(* PLC project mtcs_dome, Institute of Astronomy OntoManager 0.0.1 *)
(* stored: creationDateTime 2024-08-13T09:19:36.315732, modificationDateTime 2024-08-13T09:19:36.315732 *)

TYPE DomeParts : STRUCT
  shutter : DomeShutter;  (* Shutter mechanism *)
  rotation : DomeRotation;  (* Rotation mechanism *)
  light : DomeLight;  (* Light in dome *)
  io : DomeIO;  (* EtherCAT devices *)
  configManager : ConfigManager;  (* The config manager (to load/save/activate configuration data) *)
END_STRUCT;
END_TYPE

TYPE DomeShutterParts : STRUCT
  pumpsRelay : SimpleRelay;  (* Relay to start the pumps motors *)
  upperOpenRelay : SimpleRelay;  (* Relay to open the upper shutter panel *)
  upperCloseRelay : SimpleRelay;  (* Relay to close the upper shutter panel *)
  lowerOpenRelay : SimpleRelay;  (* Relay to open the upper shutter panel *)
  lowerCloseRelay : SimpleRelay;  (* Relay to close the upper shutter panel *)
END_STRUCT;
END_TYPE

TYPE DomeRotationParts : STRUCT
  masterAxis : AngularAxis;  (* Master axis *)
  slaveAxis : AngularAxis;  (* Slave axis *)
  drive : AX52XXDrive;  (* Dual axis drive *)
END_STRUCT;
END_TYPE

TYPE DomeLightParts : STRUCT
  switchOnRelay : SimpleRelay;  (* Relay to switch on the light *)
END_STRUCT;
END_TYPE

TYPE DomeIOParts : STRUCT
  coupler : EtherCatDevice;  (* Coupler *)
  slot1 : EtherCatDevice;  (* Slot 1 *)
  slot2 : EtherCatDevice;  (* Slot 2 *)
  slot3 : EtherCatDevice;  (* Slot 3 *)
  slot4 : EtherCatDevice;  (* Slot 4 *)
  drive : EtherCatDevice;  (* Drive *)
END_STRUCT;
END_TYPE

TYPE DomeProcesses : STRUCT
  initialize : Process;  (* Start initializing *)
  lock : Process;  (* Lock the cover *)
  unlock : Process;  (* Unlock the cover *)
  changeOperatingState : ChangeOperatingStateProcess;  (* Change the operating state (e.g. AUTO, MANUAL, ...) *)
  reset : Process;  (* Reset any errors *)
  powerOn : Process;  (* Power on the dome *)
  powerOff : Process;  (* Power off the dome *)
  syncWithAxes : Process;  (* Synchronize the dome once with the axes *)
  startTracking : Process;  (* Start tracking the axes *)
  stopTracking : Process;  (* Stop tracking the axes *)
  stop : Process;  (* Stop the rotation movement and/or tracking *)
  moveKnownPosition : DomeMoveKnownPositionProcess;  (* Move the dome to the given known position *)
END_STRUCT;
END_TYPE

TYPE DomeShutterProcesses : STRUCT
  reset : Process;  (* Reset errors *)
  open : Process;  (* Open both panels *)
  close : Process;  (* Close both panels *)
  stop : Process;  (* Stop the panels *)
  lowerOpen : Process;  (* Open the lower panel *)
  lowerClose : Process;  (* Close the lower panel *)
  upperOpen : Process;  (* Open the upper panel *)
  upperClose : Process;  (* Close the upper panel *)
END_STRUCT;
END_TYPE

TYPE DomeRotationProcesses : STRUCT
  reset : Process;  (* Reset errors *)
  stop : Process;  (* Stop the rotation *)
  moveAbsolute : DomeMoveProcess;  (* Move absolute *)
  moveRelative : DomeMoveProcess;  (* Move relative *)
  home : Process;  (* Perform a homing *)
  powerOn : Process;  (* Power on master and slave *)
  powerOff : Process;  (* Power off master and slave *)
END_STRUCT;
END_TYPE

TYPE DomeLightProcesses : STRUCT
  reset : Process;  (* Reset errors *)
  switchLightOn : Process;  (* Turn On the light in the dome *)
  switchLightOff : Process;  (* Turn Off the light in the dome *)
END_STRUCT;
END_TYPE

TYPE DomeStatuses : STRUCT
  initializationStatus : InitializationStatus;
  healthStatus : HealthStatus;
  busyStatus : BusyStatus;
  operatingStatus : OperatingStatus;
  poweredStatus : PoweredStatus;
END_STRUCT;
END_TYPE

TYPE DomeShutterStatuses : STRUCT
  apertureStatus : ApertureStatus;  (* Combined aperture status (i.e. of both panels) *)
  lowerApertureStatus : ApertureStatus;  (* Aperture status of the lower panel *)
  upperApertureStatus : ApertureStatus;  (* Aperture status of the upper panel *)
  healthStatus : HealthStatus;  (* Health status *)
  busyStatus : BusyStatus;  (* Busy status *)
END_STRUCT;
END_TYPE

TYPE DomeRotationStatuses : STRUCT
  healthStatus : HealthStatus;  (* Health status *)
  busyStatus : BusyStatus;  (* Busy status *)
  poweredStatus : PoweredStatus;  (* Powered status *)
END_STRUCT;
END_TYPE

TYPE DomeLightStatuses : STRUCT
  healthStatus : HealthStatus;  (* Health status *)
  busyStatus : BusyStatus;  (* Busy status *)
END_STRUCT;
END_TYPE

TYPE DomeIOStatuses : STRUCT
  healthStatus : HealthStatus;  (* Is the I/O in a healthy state? *)
END_STRUCT;
END_TYPE

TYPE DomeConfig : STRUCT
  shutter : DomeShutterConfig;  (* The config of the shutter mechanism *)
  rotation : DomeRotationConfig;  (* The config of the rotation system *)
  light : DomeLightConfig;  (* The config of the light in the dome *)
  maxTrackingDistance : LREAL;  (* The maximum distance between telescope and dome while tracking *)
  trackingLoopTime : LREAL;  (* Loop time, in seconds, of the tracking. *)
  knownPositions : DomeKnownPositionsConfig;  (* The known positions of the dome *)
  knownPositionTolerance : LREAL;  (* Tolerance (in degrees) to determine if the dome is at a known position *)
END_STRUCT;
END_TYPE

TYPE DomeKnownPositionConfig : STRUCT
  name : STRING;  (* The name of the position (e.g. 'PARK') *)
  position : LREAL;  (* Azimuth in degrees *)
END_STRUCT;
END_TYPE

TYPE DomeKnownPositionsConfig : STRUCT
  position0 : DomeKnownPositionConfig;  (* Known position 0 *)
  position1 : DomeKnownPositionConfig;  (* Known position 1 *)
  position2 : DomeKnownPositionConfig;  (* Known position 2 *)
  position3 : DomeKnownPositionConfig;  (* Known position 3 *)
  position4 : DomeKnownPositionConfig;  (* Known position 4 *)
  position5 : DomeKnownPositionConfig;  (* Known position 5 *)
  position6 : DomeKnownPositionConfig;  (* Known position 6 *)
  position7 : DomeKnownPositionConfig;  (* Known position 7 *)
  position8 : DomeKnownPositionConfig;  (* Known position 8 *)
  position9 : DomeKnownPositionConfig;  (* Known position 9 *)
END_STRUCT;
END_TYPE

TYPE DomeShutterConfig : STRUCT
  wirelessPolling : LREAL;  (* Polling frequency of the wireless I/O device, in seconds. Negative value = no polling. *)
  wirelessIpAddress : STRING;  (* IP address of the wireless I/O device *)
  wirelessPort : UINT;  (* Port of the wireless I/O device *)
  wirelessUnitID : USINT;  (* Unit ID the wireless I/O device *)
  wirelessTimeoutSeconds : LREAL;  (* The timeout of a single command. Does not lead to an error (yet), because we still retry. *)
  wirelessRetriesSeconds : LREAL;  (* The total timeout of the retries. If no valid data is received after this time, then we consider the shutters in error. *)
  upperEstimatedOpenTime : LREAL;  (* Estimated opening time of the upper panel, in seconds *)
  upperEstimatedCloseTime : LREAL;  (* Estimated closing time of the upper panel, in seconds *)
  lowerEstimatedOpenTime : LREAL;  (* Estimated opening time of the lower panel, in seconds *)
  lowerEstimatedCloseTime : LREAL;  (* Estimated closing time of the lower panel, in seconds *)
  lowerOpenTimeout : LREAL;  (* Opening timeout of the lower panel, in seconds *)
  lowerCloseTimeout : LREAL;  (* Closing timeout of the lower panel, in seconds *)
  upperOpenTimeout : LREAL;  (* Opening timeout of the upper panel, in seconds *)
  upperCloseTimeout : LREAL;  (* Closing timeout of the upper panel, in seconds *)
  timeAfterStop : LREAL;  (* Time to wait after a stop command, in seconds *)
END_STRUCT;
END_TYPE

TYPE DomeRotationConfig : STRUCT
  maxMovingVelocity : LREAL;  (* Maximum velocity when moving absolute or relative, in degrees per second *)
  maxMasterSlaveLag : LREAL;  (* Below this lag value (in degrees), the lag is considered not an error *)
  torqueCoefficientV : LREAL;  (* Coefficient v in 'SlaveTorque = v * MasterVelo + a * MasterAcceleration *)
  torqueCoefficientA : LREAL;  (* Coefficient a in 'SlaveTorque = v * MasterVelo + a * MasterAcceleration *)
  homePosition : LREAL;  (* Azimuth position of the home sensor, in degrees *)
  homingMoveOutOfSensorDistance : LREAL;  (* If on the sensor, move this distance, in degrees *)
  homingStage1Velocity : LREAL;  (* Velocity, in degrees per second, of the first homing stage *)
  homingStage1Timeout : LREAL;  (* Timeout of the first homing stage, in seconds *)
  homingStage2Velocity : LREAL;  (* Velocity, in degrees per second, of the second homing stage *)
  homingStage2Timeout : LREAL;  (* Timeout of the second homing stage, in seconds *)
  homingDoTwoStages : BOOL;  (* True for 2-stages homing, False for 1-stage homing. *)
  quickStopDeceleration : LREAL;  (* Quick stop deceleration, in degrees/sec2 *)
  quickStopJerk : LREAL;  (* Quick stop jerk, in degrees/sec3 *)
END_STRUCT;
END_TYPE

TYPE DomeLightConfig : STRUCT
  timeDomeLightOn : LREAL;  (* Time to keep the light on, in seconds *)
  enableDomeLight : BOOL;  (* True for enabling the control of the light *)
END_STRUCT;
END_TYPE

TYPE DomeMoveKnownPositionProcessArgs : STRUCT
  name : STRING;  (* Name of the position to move to *)
END_STRUCT;
END_TYPE

TYPE DomeMoveProcessArgs : STRUCT
  position : LREAL;  (* New absolute or relative position value in degrees *)
END_STRUCT;
END_TYPE

FUNCTION_BLOCK SM_Dome
  VAR_INPUT
    {attribute 'OPC.UA.DA' := '1'}
    {attribute 'OPC.UA.DA.Access' := '1'}
    editableConfig : DomeConfig;  (* Editable configuration of the cover *)
  END_VAR
  VAR_OUTPUT
    {attribute 'OPC.UA.DA' := '1'}
    {attribute 'OPC.UA.DA.Access' := '1'}
    actualStatus : STRING;  (* Current status description *)
    previousStatus : STRING;  (* Previous status description *)
    {attribute 'OPC.UA.DA' := '1'}
    {attribute 'OPC.UA.DA.Access' := '1'}
    config : DomeConfig;  (* Active configuration of the cover *)
    {attribute 'OPC.UA.DA' := '1'}
    {attribute 'OPC.UA.DA.Access' := '1'}
    isPoweredOffByPersonInDome : BOOL;  (* True if the dome is powered off due to a person entering the dome *)
    {attribute 'OPC.UA.DA' := '1'}
    {attribute 'OPC.UA.DA.Access' := '1'}
    isTracking : BOOL;  (* True if the dome is tracking the telescope *)
    {attribute 'OPC.UA.DA' := '1'}
    {attribute 'OPC.UA.DA.Access' := '1'}
    telescopeTargetDistance : AngularPosition;  (* Actual distance between telescope target and dome *)
    {attribute 'OPC.UA.DA' := '1'}
    {attribute 'OPC.UA.DA.Access' := '1'}
    isAtKnownPosition : BOOL;  (* True if the dome is at a known position *)
    {attribute 'OPC.UA.DA' := '1'}
    {attribute 'OPC.UA.DA.Access' := '1'}
    actualKnownPositionName : STRING;  (* Name of the known position if isAtKnownPosition is True *)
    statuses : DomeStatuses;  (* Statuses of the state machine *)
    parts : DomeParts;  (* Parts of the state machine *)
    processes : DomeProcesses;  (* Processes of the state machine *)
  END_VAR
  VAR_IN_OUT
    {attribute 'OPC.UA.DA' := '0'}
    operatorStatus : OperatorStatus;  (* Reference to the operator (observer/tech) *)
    {attribute 'OPC.UA.DA' := '0'}
    activityStatus : ActivityStatus;  (* Shared activity status *)
    {attribute 'OPC.UA.DA' := '0'}
    aziTargetPos : AngularPosition;  (* Azimuth target position of the telescope Axes *)
    {attribute 'OPC.UA.DA' := '0'}
    safetyDomeShutter : SafetyDomeShutter;  (* Reference to the dome shutter safety *)
    {attribute 'OPC.UA.DA' := '0'}
    safetyMotionBlocking : SafetyMotionBlocking;  (* Reference to the motion blocking safety *)
    {attribute 'OPC.UA.DA' := '0'}
    safetyDomeAccess : SafetyDomeAccess;  (* Reference to the dome access safety *)
  END_VAR

            parts.shutter(
    initializationStatus := statuses.initializationStatus,
    operatorStatus := operatorStatus,
    operatingStatus := statuses.operatingStatus,
    activityStatus := activityStatus,
    safety := safetyDomeShutter,
    config := config.shutter);
parts.rotation(
    initializationStatus := statuses.initializationStatus,
    operatorStatus := operatorStatus,
    operatingStatus := statuses.operatingStatus,
    config := config.rotation);
parts.light(
    initializationStatus := statuses.initializationStatus,
    operatorStatus := operatorStatus,
    operatingStatus := statuses.operatingStatus,
    activityStatus := activityStatus,
    config := config.light);
parts.io();
parts.configManager( isEnabled := operatorStatus.tech );
statuses.initializationStatus();
statuses.healthStatus(
    isGood := parts.shutter.statuses.healthStatus.isGood AND (parts.rotation.statuses.healthStatus.isGood AND (parts.light.statuses.healthStatus.isGood AND parts.io.statuses.healthStatus.isGood)),
    hasWarning := parts.shutter.statuses.healthStatus.hasWarning OR (parts.rotation.statuses.healthStatus.hasWarning OR (parts.light.statuses.healthStatus.hasWarning OR parts.io.statuses.healthStatus.hasWarning)));
statuses.busyStatus( isBusy := parts.shutter.statuses.busyStatus.busy OR parts.rotation.statuses.busyStatus.busy );
statuses.operatingStatus( superState := statuses.initializationStatus.initialized );
statuses.poweredStatus( isEnabled := parts.rotation.statuses.poweredStatus.enabled );
processes.initialize( isEnabled := (NOT(statuses.initializationStatus.locked)) AND (statuses.initializationStatus.shutdown OR (statuses.initializationStatus.initializingFailed OR statuses.initializationStatus.initialized)) );
processes.lock( isEnabled := operatorStatus.tech );
processes.unlock( isEnabled := operatorStatus.tech AND statuses.initializationStatus.locked );
processes.changeOperatingState( isEnabled := FALSE );
processes.reset( isEnabled := statuses.busyStatus.idle AND statuses.initializationStatus.initialized );
processes.powerOn( isEnabled := (NOT(statuses.initializationStatus.locked)) AND (statuses.initializationStatus.initialized AND processes.powerOn.statuses.busyStatus.idle) );
processes.powerOff( isEnabled := statuses.initializationStatus.initialized AND processes.powerOff.statuses.busyStatus.idle );
processes.syncWithAxes( isEnabled := statuses.initializationStatus.initialized AND (statuses.busyStatus.idle AND (statuses.poweredStatus.enabled AND parts.rotation.isHomed)) );
processes.startTracking( isEnabled := statuses.poweredStatus.enabled AND ((NOT(isTracking)) AND parts.rotation.isHomed) );
processes.stopTracking( isEnabled := isTracking );
processes.stop( isEnabled := statuses.busyStatus.busy OR (isTracking OR operatorStatus.tech) );
processes.moveKnownPosition( isEnabled := statuses.initializationStatus.initialized AND (statuses.busyStatus.idle AND (statuses.poweredStatus.enabled AND parts.rotation.isHomed)) );

          

{attribute 'TcRpcEnable' := '1'}
METHOD initialize : RequestResults
                  initialize := THIS^.processes.initialize.request();

                
END_METHOD

{attribute 'TcRpcEnable' := '1'}
METHOD lock : RequestResults
                  lock := THIS^.processes.lock.request();

                
END_METHOD

{attribute 'TcRpcEnable' := '1'}
METHOD unlock : RequestResults
                  unlock := THIS^.processes.unlock.request();

                
END_METHOD

{attribute 'TcRpcEnable' := '1'}
METHOD changeOperatingState : RequestResults
  VAR_INPUT
    state : OperatingStates;
  END_VAR
                  changeOperatingState := THIS^.processes.changeOperatingState.request( state := state );

                
END_METHOD

{attribute 'TcRpcEnable' := '1'}
METHOD reset : RequestResults
                  reset := THIS^.processes.reset.request();

                
END_METHOD

{attribute 'TcRpcEnable' := '1'}
METHOD powerOn : RequestResults
                  powerOn := THIS^.processes.powerOn.request();

                
END_METHOD

{attribute 'TcRpcEnable' := '1'}
METHOD powerOff : RequestResults
                  powerOff := THIS^.processes.powerOff.request();

                
END_METHOD

{attribute 'TcRpcEnable' := '1'}
METHOD syncWithAxes : RequestResults
                  syncWithAxes := THIS^.processes.syncWithAxes.request();

                
END_METHOD

{attribute 'TcRpcEnable' := '1'}
METHOD startTracking : RequestResults
                  startTracking := THIS^.processes.startTracking.request();

                
END_METHOD

{attribute 'TcRpcEnable' := '1'}
METHOD stopTracking : RequestResults
                  stopTracking := THIS^.processes.stopTracking.request();

                
END_METHOD

{attribute 'TcRpcEnable' := '1'}
METHOD stop : RequestResults
                  stop := THIS^.processes.stop.request();

                
END_METHOD

{attribute 'TcRpcEnable' := '1'}
METHOD moveKnownPosition : RequestResults
  VAR_INPUT
    name : STRING;
  END_VAR
                  moveKnownPosition := THIS^.processes.moveKnownPosition.request( name := name );

                
END_METHOD

{attribute 'TcRpcEnable' := '1'}
METHOD _log : BOOL
  VAR_INPUT
    name : STRING;  (* Name of this function block instance *)
  END_VAR
  VAR_IN_OUT
    buffer : LogBuffer;  (* Buffer to write all logging to *)
  END_VAR
  VAR
    subBuffer : LogBuffer;  (* Temporary buffer to write logging by parts (sub-statemachines) to *)
  END_VAR
                  THIS^.parts.shutter._log(
    name := 'shutter',
    buffer := subBuffer);
THIS^.parts.rotation._log(
    name := 'rotation',
    buffer := subBuffer);
THIS^.parts.light._log(
    name := 'light',
    buffer := subBuffer);
THIS^.parts.io._log(
    name := 'io',
    buffer := subBuffer);
THIS^.parts.configManager._log(
    name := 'configManager',
    buffer := subBuffer);
THIS^.processes.initialize._log(
    name := 'processes.initialize',
    buffer := subBuffer);
THIS^.processes.lock._log(
    name := 'processes.lock',
    buffer := subBuffer);
THIS^.processes.unlock._log(
    name := 'processes.unlock',
    buffer := subBuffer);
THIS^.processes.changeOperatingState._log(
    name := 'processes.changeOperatingState',
    buffer := subBuffer);
THIS^.processes.reset._log(
    name := 'processes.reset',
    buffer := subBuffer);
THIS^.processes.powerOn._log(
    name := 'processes.powerOn',
    buffer := subBuffer);
THIS^.processes.powerOff._log(
    name := 'processes.powerOff',
    buffer := subBuffer);
THIS^.processes.syncWithAxes._log(
    name := 'processes.syncWithAxes',
    buffer := subBuffer);
THIS^.processes.startTracking._log(
    name := 'processes.startTracking',
    buffer := subBuffer);
THIS^.processes.stopTracking._log(
    name := 'processes.stopTracking',
    buffer := subBuffer);
THIS^.processes.stop._log(
    name := 'processes.stop',
    buffer := subBuffer);
THIS^.processes.moveKnownPosition._log(
    name := 'processes.moveKnownPosition',
    buffer := subBuffer);
LOGGER(
    name := name,
    actualStatus := THIS^.actualStatus,
    previousStatus := THIS^.previousStatus,
    buffer := buffer,
    subBuffer := subBuffer,
    pHealthStatus := ADR(THIS^.statuses.healthStatus),
    pBusyStatus := ADR(THIS^.statuses.busyStatus));

                
END_METHOD
END_FUNCTION_BLOCK

FUNCTION_BLOCK SM_DomeShutter
  VAR_INPUT
    {attribute 'OPC.UA.DA' := '1'}
    {attribute 'OPC.UA.DA.Access' := '1'}
    lowerOpenSignal : BOOL;  (* False if the signal is not present OR if there is a communication error *)
    {attribute 'OPC.UA.DA' := '1'}
    {attribute 'OPC.UA.DA.Access' := '1'}
    lowerClosedSignal : BOOL;  (* False if the signal is not present OR if there is a communication error *)
    {attribute 'OPC.UA.DA' := '1'}
    {attribute 'OPC.UA.DA.Access' := '1'}
    upperOpenSignal : BOOL;  (* False if the signal is not present OR if there is a communication error *)
    {attribute 'OPC.UA.DA' := '1'}
    {attribute 'OPC.UA.DA.Access' := '1'}
    upperClosedSignal : BOOL;  (* False if the signal is not present OR if there is a communication error *)
    {attribute 'OPC.UA.DA' := '1'}
    {attribute 'OPC.UA.DA.Access' := '1'}
    wirelessTimeout : BOOL;  (* True if the wireless communication to the shutter signals is timing out *)
    {attribute 'OPC.UA.DA' := '1'}
    {attribute 'OPC.UA.DA.Access' := '1'}
    wirelessError : BOOL;  (* True if the wireless communication to the shutter signals is in error (other than timeout) *)
    {attribute 'OPC.UA.DA' := '1'}
    {attribute 'OPC.UA.DA.Access' := '1'}
    wirelessErrorId : UDINT;  (* The error id if wirelessError is true *)
    {attribute 'OPC.UA.DA' := '1'}
    {attribute 'OPC.UA.DA.Access' := '1'}
    wirelessData : UINT;  (* The received wireless data *)
    {attribute 'OPC.UA.DA' := '1'}
    {attribute 'OPC.UA.DA.Access' := '1'}
    upperTimeRemaining : Duration;  (* Estimated time remaining to open/close the upper panel *)
    {attribute 'OPC.UA.DA' := '1'}
    {attribute 'OPC.UA.DA.Access' := '1'}
    lowerTimeRemaining : Duration;  (* Estimated time remaining to open/close the lower panel *)
    {attribute 'OPC.UA.DA' := '1'}
    {attribute 'OPC.UA.DA.Access' := '1'}
    isLowerMonitored : BOOL;  (* TRUE if the lower shutter panel is being monitored *)
    {attribute 'OPC.UA.DA' := '1'}
    {attribute 'OPC.UA.DA.Access' := '1'}
    noOfLowerAutoClosings : INT;  (* The number of times that the lower panel has been closed automatically, by monitoring *)
    {attribute 'OPC.UA.DA' := '1'}
    {attribute 'OPC.UA.DA.Access' := '1'}
    manualOpenUpper AT %I* : BOOL;  (* Manual operation: open upper switch *)
    {attribute 'OPC.UA.DA' := '1'}
    {attribute 'OPC.UA.DA.Access' := '1'}
    manualCloseUpper AT %I* : BOOL;  (* Manual operation: close upper switch *)
    {attribute 'OPC.UA.DA' := '1'}
    {attribute 'OPC.UA.DA.Access' := '1'}
    manualOpenLower AT %I* : BOOL;  (* Manual operation: open lower switch *)
    {attribute 'OPC.UA.DA' := '1'}
    {attribute 'OPC.UA.DA.Access' := '1'}
    manualCloseLower AT %I* : BOOL;  (* Manual operation: close lower switch *)
    {attribute 'OPC.UA.DA' := '1'}
    {attribute 'OPC.UA.DA.Access' := '1'}
    manualPumpOn AT %I* : BOOL;  (* Manual operation: pump ON *)
    {attribute 'OPC.UA.DA' := '1'}
    {attribute 'OPC.UA.DA.Access' := '1'}
    automaticOperation AT %I* : BOOL;  (* TRUE if switch is on Auto, FALSE if switch is Manual *)
  END_VAR
  VAR_OUTPUT
    {attribute 'OPC.UA.DA' := '1'}
    {attribute 'OPC.UA.DA.Access' := '1'}
    actualStatus : STRING;  (* Current status description *)
    previousStatus : STRING;  (* Previous status description *)
    statuses : DomeShutterStatuses;  (* Statuses of the state machine *)
    parts : DomeShutterParts;  (* Parts of the state machine *)
    processes : DomeShutterProcesses;  (* Processes of the state machine *)
  END_VAR
  VAR_IN_OUT
    {attribute 'OPC.UA.DA' := '0'}
    initializationStatus : InitializationStatus;  (* Dome initialization status (initialized/initializing/...) *)
    {attribute 'OPC.UA.DA' := '0'}
    operatorStatus : OperatorStatus;  (* MTCS operator (observer/tech) *)
    {attribute 'OPC.UA.DA' := '0'}
    operatingStatus : OperatingStatus;  (* Dome operating status (manual/auto) *)
    {attribute 'OPC.UA.DA' := '0'}
    activityStatus : ActivityStatus;  (* Shared activity status *)
    {attribute 'OPC.UA.DA' := '0'}
    safety : SafetyDomeShutter;  (* The dome shutter safety *)
    {attribute 'OPC.UA.DA' := '0'}
    config : DomeShutterConfig;  (* The shutter config *)
  END_VAR

            parts.pumpsRelay( isEnabled := operatorStatus.tech );
parts.upperOpenRelay( isEnabled := operatorStatus.tech );
parts.upperCloseRelay( isEnabled := operatorStatus.tech );
parts.lowerOpenRelay( isEnabled := operatorStatus.tech );
parts.lowerCloseRelay( isEnabled := operatorStatus.tech );
statuses.apertureStatus(
    superState := NOT(wirelessTimeout OR wirelessError),
    isOpen := statuses.lowerApertureStatus.open AND statuses.upperApertureStatus.open,
    isClosed := statuses.lowerApertureStatus.closed AND statuses.upperApertureStatus.closed);
statuses.lowerApertureStatus(
    superState := NOT(wirelessTimeout OR wirelessError),
    isOpen := lowerOpenSignal,
    isClosed := lowerClosedSignal);
statuses.upperApertureStatus(
    superState := NOT(wirelessTimeout OR wirelessError),
    isOpen := upperOpenSignal,
    isClosed := upperClosedSignal);
statuses.healthStatus(
    isGood := (NOT(wirelessTimeout OR wirelessError)) AND (processes.reset.statuses.healthStatus.isGood AND (processes.open.statuses.healthStatus.isGood AND (processes.close.statuses.healthStatus.isGood AND (processes.stop.statuses.healthStatus.isGood AND (processes.lowerOpen.statuses.healthStatus.isGood AND (processes.lowerClose.statuses.healthStatus.isGood AND (processes.upperOpen.statuses.healthStatus.isGood AND processes.upperClose.statuses.healthStatus.isGood))))))),
    hasWarning := (processes.reset.statuses.healthStatus.hasWarning OR (processes.open.statuses.healthStatus.hasWarning OR (processes.close.statuses.healthStatus.hasWarning OR (processes.stop.statuses.healthStatus.hasWarning OR (processes.lowerOpen.statuses.healthStatus.hasWarning OR (processes.lowerClose.statuses.healthStatus.hasWarning OR (processes.upperOpen.statuses.healthStatus.hasWarning OR processes.upperClose.statuses.healthStatus.hasWarning))))))) OR ((statuses.busyStatus.idle AND statuses.lowerApertureStatus.partiallyOpen) OR ((statuses.busyStatus.idle AND statuses.upperApertureStatus.partiallyOpen) OR (NOT(automaticOperation)))));
statuses.busyStatus( isBusy := processes.reset.statuses.busyStatus.busy OR (processes.open.statuses.busyStatus.busy OR (processes.close.statuses.busyStatus.busy OR (processes.stop.statuses.busyStatus.busy OR (processes.lowerOpen.statuses.busyStatus.busy OR (processes.lowerClose.statuses.busyStatus.busy OR (processes.upperOpen.statuses.busyStatus.busy OR processes.upperClose.statuses.busyStatus.busy)))))) );
processes.reset( isEnabled := TRUE );
processes.open( isEnabled := statuses.healthStatus.isGood AND ((NOT(initializationStatus.locked)) AND (operatorStatus.tech OR (statuses.busyStatus.idle AND (initializationStatus.initialized AND (activityStatus.awake OR activityStatus.moving))))) );
processes.close( isEnabled := statuses.healthStatus.isGood AND ((NOT(initializationStatus.locked)) AND (statuses.busyStatus.idle AND initializationStatus.initialized)) );
processes.stop( isEnabled := statuses.busyStatus.busy );
processes.lowerOpen( isEnabled := processes.open.isEnabled );
processes.lowerClose( isEnabled := processes.close.isEnabled );
processes.upperOpen( isEnabled := processes.open.isEnabled );
processes.upperClose( isEnabled := processes.close.isEnabled );

          

{attribute 'TcRpcEnable' := '1'}
METHOD reset : RequestResults
                  reset := THIS^.processes.reset.request();

                
END_METHOD

{attribute 'TcRpcEnable' := '1'}
METHOD open : RequestResults
                  open := THIS^.processes.open.request();

                
END_METHOD

{attribute 'TcRpcEnable' := '1'}
METHOD close : RequestResults
                  close := THIS^.processes.close.request();

                
END_METHOD

{attribute 'TcRpcEnable' := '1'}
METHOD stop : RequestResults
                  stop := THIS^.processes.stop.request();

                
END_METHOD

{attribute 'TcRpcEnable' := '1'}
METHOD lowerOpen : RequestResults
                  lowerOpen := THIS^.processes.lowerOpen.request();

                
END_METHOD

{attribute 'TcRpcEnable' := '1'}
METHOD lowerClose : RequestResults
                  lowerClose := THIS^.processes.lowerClose.request();

                
END_METHOD

{attribute 'TcRpcEnable' := '1'}
METHOD upperOpen : RequestResults
                  upperOpen := THIS^.processes.upperOpen.request();

                
END_METHOD

{attribute 'TcRpcEnable' := '1'}
METHOD upperClose : RequestResults
                  upperClose := THIS^.processes.upperClose.request();

                
END_METHOD

{attribute 'TcRpcEnable' := '1'}
METHOD _log : BOOL
  VAR_INPUT
    name : STRING;  (* Name of this function block instance *)
  END_VAR
  VAR_IN_OUT
    buffer : LogBuffer;  (* Buffer to write all logging to *)
  END_VAR
  VAR
    subBuffer : LogBuffer;  (* Temporary buffer to write logging by parts (sub-statemachines) to *)
  END_VAR
                  THIS^.parts.pumpsRelay._log(
    name := 'pumpsRelay',
    buffer := subBuffer);
THIS^.parts.upperOpenRelay._log(
    name := 'upperOpenRelay',
    buffer := subBuffer);
THIS^.parts.upperCloseRelay._log(
    name := 'upperCloseRelay',
    buffer := subBuffer);
THIS^.parts.lowerOpenRelay._log(
    name := 'lowerOpenRelay',
    buffer := subBuffer);
THIS^.parts.lowerCloseRelay._log(
    name := 'lowerCloseRelay',
    buffer := subBuffer);
THIS^.processes.reset._log(
    name := 'processes.reset',
    buffer := subBuffer);
THIS^.processes.open._log(
    name := 'processes.open',
    buffer := subBuffer);
THIS^.processes.close._log(
    name := 'processes.close',
    buffer := subBuffer);
THIS^.processes.stop._log(
    name := 'processes.stop',
    buffer := subBuffer);
THIS^.processes.lowerOpen._log(
    name := 'processes.lowerOpen',
    buffer := subBuffer);
THIS^.processes.lowerClose._log(
    name := 'processes.lowerClose',
    buffer := subBuffer);
THIS^.processes.upperOpen._log(
    name := 'processes.upperOpen',
    buffer := subBuffer);
THIS^.processes.upperClose._log(
    name := 'processes.upperClose',
    buffer := subBuffer);
LOGGER(
    name := name,
    actualStatus := THIS^.actualStatus,
    previousStatus := THIS^.previousStatus,
    buffer := buffer,
    subBuffer := subBuffer,
    pHealthStatus := ADR(THIS^.statuses.healthStatus),
    pBusyStatus := ADR(THIS^.statuses.busyStatus));

                
END_METHOD
END_FUNCTION_BLOCK

FUNCTION_BLOCK SM_DomeRotation
  VAR_OUTPUT
    {attribute 'OPC.UA.DA' := '1'}
    {attribute 'OPC.UA.DA.Access' := '1'}
    actualStatus : STRING;  (* Current status description *)
    previousStatus : STRING;  (* Previous status description *)
    {attribute 'OPC.UA.DA' := '1'}
    {attribute 'OPC.UA.DA.Access' := '1'}
    actPos : AngularPosition;  (* The actual position (same as parts.masterAxis!) *)
    {attribute 'OPC.UA.DA' := '1'}
    {attribute 'OPC.UA.DA.Access' := '1'}
    actVelo : AngularVelocity;  (* The actual velocity (same as parts.masterAxis!) *)
    {attribute 'OPC.UA.DA' := '1'}
    {attribute 'OPC.UA.DA.Access' := '1'}
    actTorqueMaster : Torque;  (* The actual torque on the telescope axis by the master motor *)
    {attribute 'OPC.UA.DA' := '1'}
    {attribute 'OPC.UA.DA.Access' := '1'}
    actTorqueSlave : Torque;  (* The actual torque on the telescope axis by the slave motor *)
    {attribute 'OPC.UA.DA' := '1'}
    {attribute 'OPC.UA.DA.Access' := '1'}
    masterSlaveLag : AngularPosition;  (* masterAxis.actPos - slaveAxis.actPos *)
    {attribute 'OPC.UA.DA' := '1'}
    {attribute 'OPC.UA.DA.Access' := '1'}
    masterSlaveLagError : BOOL;  (* (ABS(masterSlaveLag) >= config.maxMasterSlaveLag) AND isHomed AND poweredOn *)
    {attribute 'OPC.UA.DA' := '1'}
    {attribute 'OPC.UA.DA.Access' := '1'}
    homingSensorSignal : BOOL;  (* True = at home position *)
    {attribute 'OPC.UA.DA' := '1'}
    {attribute 'OPC.UA.DA.Access' := '1'}
    isHomed : BOOL;  (* True if homing was done *)
    statuses : DomeRotationStatuses;  (* Statuses of the state machine *)
    parts : DomeRotationParts;  (* Parts of the state machine *)
    processes : DomeRotationProcesses;  (* Processes of the state machine *)
  END_VAR
  VAR_IN_OUT
    {attribute 'OPC.UA.DA' := '0'}
    initializationStatus : InitializationStatus;  (* Reference to the MTCS initialization status *)
    {attribute 'OPC.UA.DA' := '0'}
    operatorStatus : OperatorStatus;  (* Reference to the MTCS operator status *)
    {attribute 'OPC.UA.DA' := '0'}
    operatingStatus : OperatingStatus;  (* Reference to the Dome operating status *)
    {attribute 'OPC.UA.DA' := '0'}
    config : DomeRotationConfig;  (* Reference to the rotation config *)
  END_VAR

            parts.masterAxis( isEnabled := (NOT(initializationStatus.locked)) AND operatorStatus.tech );
parts.slaveAxis( isEnabled := (NOT(initializationStatus.locked)) AND operatorStatus.tech );
parts.drive( isEnabled := (NOT(initializationStatus.locked)) AND operatorStatus.tech );
statuses.healthStatus(
    isGood := (parts.masterAxis.statuses.healthStatus.isGood AND (parts.slaveAxis.statuses.healthStatus.isGood AND (parts.drive.statuses.healthStatus.isGood AND (processes.reset.statuses.healthStatus.isGood AND processes.stop.statuses.healthStatus.isGood)))) AND ((NOT(masterSlaveLagError)) AND (isHomed OR (NOT(initializationStatus.initialized)))),
    hasWarning := parts.masterAxis.statuses.healthStatus.hasWarning OR (parts.slaveAxis.statuses.healthStatus.hasWarning OR (parts.drive.statuses.healthStatus.hasWarning OR (processes.reset.statuses.healthStatus.hasWarning OR processes.stop.statuses.healthStatus.hasWarning))));
statuses.busyStatus( isBusy := parts.masterAxis.statuses.busyStatus.busy OR (parts.slaveAxis.statuses.busyStatus.busy OR (parts.drive.statuses.busyStatus.busy OR (processes.reset.statuses.busyStatus.busy OR processes.stop.statuses.busyStatus.busy))) );
statuses.poweredStatus( isEnabled := parts.masterAxis.statuses.poweredStatus.enabled AND parts.slaveAxis.statuses.poweredStatus.enabled );
processes.reset( isEnabled := statuses.busyStatus.idle );
processes.stop( isEnabled := statuses.busyStatus.busy OR operatorStatus.tech );
processes.moveAbsolute( isEnabled := statuses.busyStatus.idle AND statuses.poweredStatus.enabled );
processes.moveRelative( isEnabled := processes.moveAbsolute.isEnabled );
processes.home( isEnabled := processes.moveAbsolute.isEnabled );
processes.powerOn( isEnabled := (NOT(initializationStatus.locked)) AND statuses.busyStatus.idle );
processes.powerOff( isEnabled := statuses.busyStatus.idle );

          

{attribute 'TcRpcEnable' := '1'}
METHOD reset : RequestResults
                  reset := THIS^.processes.reset.request();

                
END_METHOD

{attribute 'TcRpcEnable' := '1'}
METHOD stop : RequestResults
                  stop := THIS^.processes.stop.request();

                
END_METHOD

{attribute 'TcRpcEnable' := '1'}
METHOD moveAbsolute : RequestResults
  VAR_INPUT
    position : LREAL;
  END_VAR
                  moveAbsolute := THIS^.processes.moveAbsolute.request( position := position );

                
END_METHOD

{attribute 'TcRpcEnable' := '1'}
METHOD moveRelative : RequestResults
  VAR_INPUT
    position : LREAL;
  END_VAR
                  moveRelative := THIS^.processes.moveRelative.request( position := position );

                
END_METHOD

{attribute 'TcRpcEnable' := '1'}
METHOD home : RequestResults
                  home := THIS^.processes.home.request();

                
END_METHOD

{attribute 'TcRpcEnable' := '1'}
METHOD powerOn : RequestResults
                  powerOn := THIS^.processes.powerOn.request();

                
END_METHOD

{attribute 'TcRpcEnable' := '1'}
METHOD powerOff : RequestResults
                  powerOff := THIS^.processes.powerOff.request();

                
END_METHOD

{attribute 'TcRpcEnable' := '1'}
METHOD _log : BOOL
  VAR_INPUT
    name : STRING;  (* Name of this function block instance *)
  END_VAR
  VAR_IN_OUT
    buffer : LogBuffer;  (* Buffer to write all logging to *)
  END_VAR
  VAR
    subBuffer : LogBuffer;  (* Temporary buffer to write logging by parts (sub-statemachines) to *)
  END_VAR
                  THIS^.parts.masterAxis._log(
    name := 'masterAxis',
    buffer := subBuffer);
THIS^.parts.slaveAxis._log(
    name := 'slaveAxis',
    buffer := subBuffer);
THIS^.parts.drive._log(
    name := 'drive',
    buffer := subBuffer);
THIS^.processes.reset._log(
    name := 'processes.reset',
    buffer := subBuffer);
THIS^.processes.stop._log(
    name := 'processes.stop',
    buffer := subBuffer);
THIS^.processes.moveAbsolute._log(
    name := 'processes.moveAbsolute',
    buffer := subBuffer);
THIS^.processes.moveRelative._log(
    name := 'processes.moveRelative',
    buffer := subBuffer);
THIS^.processes.home._log(
    name := 'processes.home',
    buffer := subBuffer);
THIS^.processes.powerOn._log(
    name := 'processes.powerOn',
    buffer := subBuffer);
THIS^.processes.powerOff._log(
    name := 'processes.powerOff',
    buffer := subBuffer);
LOGGER(
    name := name,
    actualStatus := THIS^.actualStatus,
    previousStatus := THIS^.previousStatus,
    buffer := buffer,
    subBuffer := subBuffer,
    pHealthStatus := ADR(THIS^.statuses.healthStatus),
    pBusyStatus := ADR(THIS^.statuses.busyStatus));

                
END_METHOD
END_FUNCTION_BLOCK

FUNCTION_BLOCK SM_DomeLight
  VAR_INPUT
    {attribute 'OPC.UA.DA' := '1'}
    {attribute 'OPC.UA.DA.Access' := '1'}
    switchOnSignal : BOOL;  (* True if the light must be switched ON *)
    {attribute 'OPC.UA.DA' := '1'}
    {attribute 'OPC.UA.DA.Access' := '1'}
    switchOnInput AT %I* : BOOL;  (* External operation: switch ON *)
    {attribute 'OPC.UA.DA' := '1'}
    {attribute 'OPC.UA.DA.Access' := '1'}
    isDomeLightON : BOOL;  (* Flag to indicate if dome light is ON or OFF *)
  END_VAR
  VAR_OUTPUT
    {attribute 'OPC.UA.DA' := '1'}
    {attribute 'OPC.UA.DA.Access' := '1'}
    actualStatus : STRING;  (* Current status description *)
    previousStatus : STRING;  (* Previous status description *)
    statuses : DomeLightStatuses;  (* Statuses of the state machine *)
    parts : DomeLightParts;  (* Parts of the state machine *)
    processes : DomeLightProcesses;  (* Processes of the state machine *)
  END_VAR
  VAR_IN_OUT
    {attribute 'OPC.UA.DA' := '0'}
    initializationStatus : InitializationStatus;  (* Dome initialization status (initialized/initializing/...) *)
    {attribute 'OPC.UA.DA' := '0'}
    operatorStatus : OperatorStatus;  (* MTCS operator (observer/tech) *)
    {attribute 'OPC.UA.DA' := '0'}
    operatingStatus : OperatingStatus;  (* Dome operating status (manual/auto) *)
    {attribute 'OPC.UA.DA' := '0'}
    activityStatus : ActivityStatus;  (* Shared activity status *)
    {attribute 'OPC.UA.DA' := '0'}
    config : DomeLightConfig;  (* The light config *)
  END_VAR

            parts.switchOnRelay( isEnabled := operatorStatus.tech );
statuses.healthStatus(
    isGood := processes.reset.statuses.healthStatus.isGood AND (processes.switchLightOn.statuses.healthStatus.isGood AND processes.switchLightOff.statuses.healthStatus.isGood),
    hasWarning := isDomeLightON OR (processes.reset.statuses.healthStatus.hasWarning OR (processes.switchLightOn.statuses.healthStatus.hasWarning OR processes.switchLightOff.statuses.healthStatus.hasWarning)));
statuses.busyStatus( isBusy := processes.reset.statuses.busyStatus.busy OR (processes.switchLightOn.statuses.busyStatus.busy OR processes.switchLightOff.statuses.busyStatus.busy) );
processes.reset( isEnabled := TRUE );
processes.switchLightOn( isEnabled := TRUE );
processes.switchLightOff( isEnabled := TRUE );

          

{attribute 'TcRpcEnable' := '1'}
METHOD reset : RequestResults
                  reset := THIS^.processes.reset.request();

                
END_METHOD

{attribute 'TcRpcEnable' := '1'}
METHOD switchLightOn : RequestResults
                  switchLightOn := THIS^.processes.switchLightOn.request();

                
END_METHOD

{attribute 'TcRpcEnable' := '1'}
METHOD switchLightOff : RequestResults
                  switchLightOff := THIS^.processes.switchLightOff.request();

                
END_METHOD

{attribute 'TcRpcEnable' := '1'}
METHOD _log : BOOL
  VAR_INPUT
    name : STRING;  (* Name of this function block instance *)
  END_VAR
  VAR_IN_OUT
    buffer : LogBuffer;  (* Buffer to write all logging to *)
  END_VAR
  VAR
    subBuffer : LogBuffer;  (* Temporary buffer to write logging by parts (sub-statemachines) to *)
  END_VAR
                  THIS^.parts.switchOnRelay._log(
    name := 'switchOnRelay',
    buffer := subBuffer);
THIS^.processes.reset._log(
    name := 'processes.reset',
    buffer := subBuffer);
THIS^.processes.switchLightOn._log(
    name := 'processes.switchLightOn',
    buffer := subBuffer);
THIS^.processes.switchLightOff._log(
    name := 'processes.switchLightOff',
    buffer := subBuffer);
LOGGER(
    name := name,
    actualStatus := THIS^.actualStatus,
    previousStatus := THIS^.previousStatus,
    buffer := buffer,
    subBuffer := subBuffer,
    pHealthStatus := ADR(THIS^.statuses.healthStatus),
    pBusyStatus := ADR(THIS^.statuses.busyStatus));

                
END_METHOD
END_FUNCTION_BLOCK

FUNCTION_BLOCK SM_DomeIO
  VAR_OUTPUT
    {attribute 'OPC.UA.DA' := '1'}
    {attribute 'OPC.UA.DA.Access' := '1'}
    actualStatus : STRING;  (* Current status description *)
    previousStatus : STRING;  (* Previous status description *)
    statuses : DomeIOStatuses;  (* Statuses of the state machine *)
    parts : DomeIOParts;  (* Parts of the state machine *)
  END_VAR

            parts.coupler(
    id := '110A1',
    typeId := 'EK1101');
parts.slot1(
    id := '111A0',
    typeId := 'ES1008');
parts.slot2(
    id := '112A0',
    typeId := 'EL2904');
parts.slot3(
    id := '112A5',
    typeId := 'EL2904');
parts.slot4(
    id := 'DO:RO1',
    typeId := 'EL2622');
parts.drive(
    id := '10U1',
    typeId := 'AX5206');
statuses.healthStatus( isGood := parts.coupler.statuses.healthStatus.isGood AND (parts.slot1.statuses.healthStatus.isGood AND (parts.slot2.statuses.healthStatus.isGood AND (parts.slot3.statuses.healthStatus.isGood AND (parts.slot4.statuses.healthStatus.isGood AND parts.drive.statuses.healthStatus.isGood)))) );

          

{attribute 'TcRpcEnable' := '1'}
METHOD _log : BOOL
  VAR_INPUT
    name : STRING;  (* Name of this function block instance *)
  END_VAR
  VAR_IN_OUT
    buffer : LogBuffer;  (* Buffer to write all logging to *)
  END_VAR
  VAR
    subBuffer : LogBuffer;  (* Temporary buffer to write logging by parts (sub-statemachines) to *)
  END_VAR
                  THIS^.parts.coupler._log(
    name := 'coupler',
    buffer := subBuffer);
THIS^.parts.slot1._log(
    name := 'slot1',
    buffer := subBuffer);
THIS^.parts.slot2._log(
    name := 'slot2',
    buffer := subBuffer);
THIS^.parts.slot3._log(
    name := 'slot3',
    buffer := subBuffer);
THIS^.parts.slot4._log(
    name := 'slot4',
    buffer := subBuffer);
THIS^.parts.drive._log(
    name := 'drive',
    buffer := subBuffer);
LOGGER(
    name := name,
    actualStatus := THIS^.actualStatus,
    previousStatus := THIS^.previousStatus,
    buffer := buffer,
    subBuffer := subBuffer,
    pHealthStatus := ADR(THIS^.statuses.healthStatus));

                
END_METHOD
END_FUNCTION_BLOCK

FUNCTION_BLOCK DomeMoveKnownPositionProcess EXTENDS BaseProcess
  VAR_INPUT
    {attribute 'OPC.UA.DA' := '1'}
    set : DomeMoveKnownPositionProcessArgs;  (* Arguments to be set, before writing do_request TRUE *)
  END_VAR
  VAR_OUTPUT
    {attribute 'OPC.UA.DA' := '1'}
    {attribute 'OPC.UA.DA.Access' := '1'}
    get : DomeMoveKnownPositionProcessArgs;  (* Arguments in use by the process, if do_request was accepted *)
  END_VAR

            IF do_request THEN
    do_request_result := request( name := set.name );
    do_request := FALSE;
END_IF;
SUPER^();

          

{attribute 'TcRpcEnable' := '1'}
METHOD start
  VAR_INPUT
    name : STRING;  (* Name of the position to move to *)
  END_VAR
                  THIS^.get.name := name;
THIS^.statuses.busyStatus( isBusy := TRUE );
THIS^.statuses.healthStatus( isGood := TRUE );

                
END_METHOD

{attribute 'TcRpcEnable' := '1'}
METHOD request : RequestResults
  VAR_INPUT
    name : STRING;  (* Name of the position to move to *)
  END_VAR
                  IF THIS^.statuses.enabledStatus.enabled THEN
    request := RequestResults.ACCEPTED;
    THIS^.start( name := name );
ELSE
    request := RequestResults.REJECTED;
END_IF;

                
END_METHOD
END_FUNCTION_BLOCK

FUNCTION_BLOCK DomeMoveProcess EXTENDS BaseProcess
  VAR_INPUT
    {attribute 'OPC.UA.DA' := '1'}
    set : DomeMoveProcessArgs;  (* Arguments to be set, before writing do_request TRUE *)
  END_VAR
  VAR_OUTPUT
    {attribute 'OPC.UA.DA' := '1'}
    {attribute 'OPC.UA.DA.Access' := '1'}
    get : DomeMoveProcessArgs;  (* Arguments in use by the process, if do_request was accepted *)
  END_VAR

            IF do_request THEN
    do_request_result := request( position := set.position );
    do_request := FALSE;
END_IF;
SUPER^();

          

{attribute 'TcRpcEnable' := '1'}
METHOD start
  VAR_INPUT
    position : LREAL;  (* New absolute or relative position value in degrees *)
  END_VAR
                  THIS^.get.position := position;
THIS^.statuses.busyStatus( isBusy := TRUE );
THIS^.statuses.healthStatus( isGood := TRUE );

                
END_METHOD

{attribute 'TcRpcEnable' := '1'}
METHOD request : RequestResults
  VAR_INPUT
    position : LREAL;  (* New absolute or relative position value in degrees *)
  END_VAR
                  IF THIS^.statuses.enabledStatus.enabled THEN
    request := RequestResults.ACCEPTED;
    THIS^.start( position := position );
ELSE
    request := RequestResults.REJECTED;
END_IF;

                
END_METHOD
END_FUNCTION_BLOCK
